FUNCTION_BLOCK INTERNAL FB_Base_Test EXTENDS FB_Base

SUPER^();

METHOD PUBLIC Init : BOOL
VAR_INPUT
	nId				: UINT ; // Identification number of object
	nParentId		: UINT ; // Id of higher level if applicable (0 = no parent)
	eComponentType	: E_ComponentTypes ; // Component or function type
END_VAR
// Every FB_Base instance is expected to have an Init method that calls ExecIdentifyDevice. 
// This Init method will have at least the nId and nParentId inputs.
// The eComponentType input is optional (can be hardcoded in the Init method, for example see FB_Step).
// It might also have additional inputs (changing the method signature) therefore it is not declared in FB_Base.
ExecIdentifyDevice(nId,	nParentId,	eComponentType);
END_METHOD

END_FUNCTION_BLOCK

(* stored: Version 1.1.0.1, ProductVersion 3.1.4024.11
   POU FB_Base_Test: Id {2de4065a-81b2-40da-80ee-7c5f2731ebce}, SpecialFunc None
   Method Init: Id {99c2bc24-3576-4200-a311-0977cdb2ff4a} *)
